FUNCTION Function_SettingCarLight : BOOL
VAR_INPUT
	ColorCarLight : INT; // 0 for Red, 1 for Green
    
END_VAR
VAR
END_VAR

// Set the light state
CASE ColorCarLight OF
    0:  // Red
        GVl.PedestrianLightRed := TRUE;
        GVL.PedestrianLightGreen := FALSE;
    
    1:  // Green
        GVL.PedestrianLightRed := FALSE;
        GVL.PedestrianLightGreen := TRUE;
END_CASE;

Function_SettingPedestrianLight := TRUE;

END_FUNCTION

(* stored: Version 1.1.0.1, ProductVersion 3.1.4024.12
   POU Function_SettingCarLight: Id {7834f468-6cf6-42b0-a0ce-ed52745fb4a3}, SpecialFunc None *)
